Staubli VAL3: chkIsFileExsit.pgx

program chkIsFileExsit(string x_sFileName, string x_sTargetFolder, bool& x_bRes)
  local num l_ni
begin
  //检查文件x_sFileName在目标文件夹中x_sTargetFolder是否存在
  x_bRes=false
  resize(sFileTemp,1,1)
  sFileTemp[0]=""
  if (libList(x_sTargetFolder,sFileTemp)==false)
    return
  endIf
  //
  for l_ni=0 to size(sFileTemp)-1
    if x_sFileName==sFileTemp[l_ni]
      x_bRes=true
      return
    endIf
  endFor

end
